Staubli VAL3: TEACH.dtx

mdesc mNomSpeed
num nApproIndex
num nCutIndex
num nLeaveIndex
public num nPointType
string sSItem
public num nTrajIndex
public string sMess
num nCutMc
bool bPowerFlag
bool bFirstTeach
num nTeachAction
bool bSyc
public num n500Count
num nPartID
bool bSaveTxt
bool bCheckAxisSafte
num nCursonIndex
num nAxisSpeed
